FUNCTION_BLOCK MoveRelativeTask EXTENDS TcoCore.TcoTask IMPLEMENTS IAxisIAI
VAR
    {attribute addProperty Name "<#Distance#>"}
    _distance : REAL;
    {attribute addProperty Name "<#Positionierbereich in mm#>"}
    _positionBand : REAL := 0.1;
    {attribute addProperty Name "<#Geschwindigkeit in mm/s#>"}
    _velocity : UINT := 10;
    {attribute addProperty Name "<#Beschleunigung (0 - 100)#>"}
    _acceleration : UINT := 10;
    {attribute addProperty Name "<#Schubstrombegrenzung#>"}
    _pushCurrentLimit : USINT := 10;
    _doneTrig         : R_TRIG;
    _move             : BOOL := TRUE;
    _targetDest       : REAL;
    _actPos           : REAL;
    _executeTr        : R_TRIG;
END_VAR

THIS^.Enabled := NOT DriveRef.HaltTask.Busy AND NOT DriveRef.MoveAbsoluteTask.Busy AND NOT DriveRef.HomeTask.Busy;

_executeTr(CLK := Execute());

IF Execute() THEN
    DriveRef.PlcToDrive.ControlSignal.INC := TRUE;
    DriveRef.PlcToDrive.Accelerartion     := _acceleration;
    //for Visu
    DriveRef.PlcToDrive.PositioningBand := REAL_TO_DINT((_positionBand * 100));
    DriveRef.PlcToDrive.TargetPosition  := REAL_TO_DINT((_distance * 100));

    IF _executeTr.Q THEN
        _targetDest                            := DriveRef.AxisStatus.ActPos + _distance;
        DriveRef.PlcToDrive.ControlSignal.CSTR := TRUE;
    END_IF

    DriveRef.PlcToDrive.Velocity := _velocity;
    _actPos                      := DriveRef.AxisStatus.ActPos;

    IF THIS^.ElapsedTime >= T#20MS THEN
        IF (ABS(_targetDest - DriveRef.AxisStatus.ActPos) <= _positionBand) THEN
            DoneWhen(TRUE);
            DriveRef.PlcToDrive.ControlSignal.CSTR := FALSE;
        END_IF
    END_IF

    ThrowWhen(driveRef.AxisStatus.Error);
END_IF

PROPERTY DriveRef : REFERENCE TO AxisIAI
GET
VAR
    _drive : POINTER TO AxisIAI;
END_VAR
IF __QUERYPOINTER(THIS^._ParentObject, _drive) THEN
    DriveRef REF= _drive^;
END_IF
END_GET
END_PROPERTY

METHOD PUBLIC FB_init : BOOL
VAR_INPUT
    bInitRetains : BOOL; // if TRUE, the retain variables are initialized (warm start / cold start)
    bInCopyCode  : BOOL; // if TRUE, the instance afterwards gets moved into the copy code (online change)
    ParentObject : ITcoObject;
END_VAR
SUPER^.FB_init(bInitRetains := bInitRetains, bInCopyCode := bInCopyCode, ParentObject := ParentObject);
END_METHOD

METHOD INTERNAL InvokeWithParams : ITcoTaskStatus
VAR_INPUT
    Distance         : REAL;
    PositionBand     : REAL;
    Velocity         : UINT;
    Acceleration     : UINT;
    PushCurrentLimit : USINT;
END_VAR
_distance         := Distance;
_positionBand     := PositionBand;
_velocity         := Velocity;
_acceleration     := Acceleration;
_pushCurrentLimit := PushCurrentLimit;
InvokeWithParams  := THIS^.Invoke();
END_METHOD

(*~
    <docu>
        <summary>
            Executes when task is aborted.
        </summary>
    </docu>
~*)
METHOD PROTECTED OnAbort
DriveRef.PlcToDrive.ControlSignal.CSTR      := FALSE;
THIS^.DriveRef.AxisStatus.HasBeenStopped    := TRUE;
THIS^.DriveRef.PlcToDrive.ControlSignal.RES := TRUE;

//SUPER^.Restore();
//_mcMoveAbsolute(Axis := _axisRef, Execute := FALSE);
END_METHOD

(*~
    <docu>
        <summary>
            Executes when task reaches the ```Done``` state .
        </summary>
    </docu>
~*)
METHOD PROTECTED OnDone
//DriveRef.PlcToDrive.ControlSignal.CSTR := FALSE;
//DriveRef.Restore();
END_METHOD

(*~
    <docu>
        <summary>
            Executes when task reaches the ```Error``` state.
            <para>
                Do not confuse with <see cref="PlcDocu.TcoCore.TcoTask.WhileError()"/>, that is called cyclically until '''Error''' state is left.
            </para>
        </summary>
    </docu>
~*)
METHOD PROTECTED OnError
DriveRef.PlcToDrive.ControlSignal.CSTR := FALSE;
DriveRef.SetErrorID(DriveRef.AxisStatus.ErrorId);
END_METHOD

(*~
    <docu>
        <summary>
            Restores this instance to the Ready state. Can be called explicitly or from within one of the restore mechanisms.
            <para>
                See also <see cref="PlcDocu.TcoCore.TcoTask.AutoRestorable()"/>
            </para>
        </summary>
    </docu>
~*)
METHOD Restore : ITcoRestorable
DriveRef.PlcToDrive.ControlSignal.STP  := FALSE;
DriveRef.PlcToDrive.ControlSignal.CSTR := FALSE;
SUPER^.Restore();
END_METHOD

END_FUNCTION_BLOCK

(* stored: Version 1.1.0.1, ProductVersion 3.1.4024.12
   POU MoveRelativeTask: Id {6b40abe1-1f21-4b5b-b4cb-337e0b9b5a11}, SpecialFunc None
   Property DriveRef: Id {d458cfe2-d348-4efb-b286-b2ed0e468df7}
   Get Get: Id {d93cabb7-afe3-4e4d-9c1e-1a4adde8b713}
   Method FB_init: Id {6a3c7e98-e4d6-48f0-bcfd-36bcc39ed815}
   Method InvokeWithParams: Id {c1772997-0025-4d49-929b-7ac1dd8583bb}
   Method OnAbort: Id {72f75a24-03af-4cae-b95f-265b921e83f1}
   Method OnDone: Id {979fccc6-8b40-4523-a5e3-0f9d19d96a4e}
   Method OnError: Id {c460b444-d453-47e9-93b8-012d592f689a}
   Method Restore: Id {2940ea44-6390-4b80-9fe6-46bcd75bcbf2} *)
